FUNCTION_BLOCK FB_FieldCodecSint32 IMPLEMENTS I_FieldCodec
VAR_INPUT
END_VAR
VAR_OUTPUT
END_VAR
VAR
    nValue : DINT;
END_VAR

METHOD IsPackedRepeatedField : BOOL
VAR_INPUT
	nTag	: UDINT;
END_VAR
IsPackedRepeatedField := F_IsPackedRepeatedField(nTag);
END_METHOD


METHOD ValueReader : HRESULT
VAR_IN_OUT CONSTANT
	aBuffer	: ARRAY [*] OF BYTE;
END_VAR
VAR_IN_OUT
	stState	: ST_ParserInternalState;
END_VAR
VAR_OUTPUT
	anyOut	: T_Any;
END_VAR
VAR
    nTmp : UDINT;
END_VAR

ValueReader := F_ParseRawVarint32(aBuffer, stState, nTmp);
IF FAILED(ValueReader) THEN
    RETURN;
END_IF
nValue := F_DecodeZigZag32(nTmp);
anyOut := F_ToAnyType(anyArg:= nValue);
END_METHOD

{warning 'Add method implementation '}
{attribute 'analysis' := '-33'}
METHOD ValueWriter : HRESULT
VAR_IN_OUT
	aBuffer	: ARRAY [*] OF BYTE;
END_VAR
VAR_IN_OUT
	stState	: ST_WriterInternalState;
END_VAR
VAR_INPUT
	anyIn	: ANY;
END_VAR
END_METHOD

END_FUNCTION_BLOCK

(* stored: Version 1.1.0.1
   POU FB_FieldCodecSint32: Id {5872bbd0-7f0f-48ad-9c30-e5bb23d85c6b}, SpecialFunc None
   Method IsPackedRepeatedField: Id {495b96ec-f670-4571-942b-2d9493d39e45}
   Method ValueReader: Id {0fb52bb4-2627-4e4a-8cf4-f8046717ea94}
   Method ValueWriter: Id {0f7622f3-c0bf-441a-92f1-2aafa8694ea1} *)
